KUKA KRL program: makro340.src

&ACCESS RVO2
&COMMENT GREIFER INIT
&PARAM TEMPLATE = C:\KRC\Roboter\Template\makrovorgabe.src
&PARAM TPVW_VERSION = 8.1.8
&PARAM EDITMASK = Makro999[0-999]
DEFFCT INT MAKRO340(ADV :IN)
   ;FOLD Makro Anfang ;%{PSE}%MKUKATPVW
      BOOL ADV
      ; interface to basic routines
      EXT  BAS (BAS_COMMAND  :IN,REAL  :IN )
      ; interface to VW-standard routines
      EXT VW (VW_COMMAND:IN, BOOL: IN, REAL:IN, REAL:IN, REAL:IN, REAL:IN, BOOL :IN, E6POS :IN )
      ; interface select routine
      EXTFCT INT  SELECT (SUBTYPE  :IN,INT  :IN,BOOL  :IN,ARI_TYP  :IN,INT  :IN,BOOL_TYP  :IN,INT  :IN,BOOL  :IN)
      SPS_N=-1
      ;FOLD ;%{H} %MKUKATPVW
      IF VARSTATE ("ADV") <> #INITIALIZED THEN
         ADV=FALSE
      ENDIF
      IF (NOT ADV) THEN
      ;ENDFOLD
   ;ENDFOLD
   ;FOLD -- Greifer Initialisierung -- ;%{E}%MKUKATPVW %CVW_COM %VCOMMENT %P 2:-- Greifer Initialisierung --, 3: VW_COMMENT
   ;ENDFOLD
   ;FOLD -- KS24 -- ;%{E}%MKUKATPVW %CVW_COM %VCOMMENT %P 2:-- KS24 --, 3: VW_COMMENT
   ;ENDFOLD
   ;FOLD -- Version: 01 -- ;%{E}%MKUKATPVW %CVW_COM %VCOMMENT %P 2:-- Version: 01 --, 3: VW_COMMENT
   ;ENDFOLD
   ;FOLD -- Stand: 001 -- ;%{E}%MKUKATPVW %CVW_COM %VCOMMENT %P 2:-- Stand: 001 --, 3: VW_COMMENT
   ;ENDFOLD
   ;FOLD -- letzte Aenderung 11.06.2014 PK -- ;%{E}%MKUKATPVW %CVW_COM %VCOMMENT %P 2:-- letzte Aenderung 11.06.2014 PK --, 3: VW_COMMENT
   ;ENDFOLD
   ;FOLD -- Vorwahl Spanngruppen AUS -- ;%{E}%MKUKATPVW %CVW_COM %VCOMMENT %P 2:-- Vorwahl Spanngruppen AUS --, 3: VW_COMMENT
   ;ENDFOLD
   ;FOLD F1 = AUS ;%{E}%MKUKATPVW %CVW_SPS %VBOASG %P 2:F1 = AUS, 3: BOASG
      $FLAG[1] = FALSE
   ;ENDFOLD
   ;FOLD F2 = AUS ;%{E}%MKUKATPVW %CVW_SPS %VBOASG %P 2:F2 = AUS, 3: BOASG
      $FLAG[2] = FALSE
   ;ENDFOLD
   ;FOLD F3 = AUS ;%{E}%MKUKATPVW %CVW_SPS %VBOASG %P 2:F3 = AUS, 3: BOASG
      $FLAG[3] = FALSE
   ;ENDFOLD
   ;FOLD F4 = AUS ;%{E}%MKUKATPVW %CVW_SPS %VBOASG %P 2:F4 = AUS, 3: BOASG
      $FLAG[4] = FALSE
   ;ENDFOLD
   ;FOLD F5 = AUS ;%{E}%MKUKATPVW %CVW_SPS %VBOASG %P 2:F5 = AUS, 3: BOASG
      $FLAG[5] = FALSE
   ;ENDFOLD
   ;FOLD F6 = AUS ;%{E}%MKUKATPVW %CVW_SPS %VBOASG %P 2:F6 = AUS, 3: BOASG
      $FLAG[6] = FALSE
   ;ENDFOLD
   ;FOLD F7 = AUS ;%{E}%MKUKATPVW %CVW_SPS %VBOASG %P 2:F7 = AUS, 3: BOASG
      $FLAG[7] = FALSE
   ;ENDFOLD
   ;FOLD F8 = AUS ;%{E}%MKUKATPVW %CVW_SPS %VBOASG %P 2:F8 = AUS, 3: BOASG
      $FLAG[8] = FALSE
   ;ENDFOLD
   ;FOLD F9 = AUS ;%{E}%MKUKATPVW %CVW_SPS %VBOASG %P 2:F9 = AUS, 3: BOASG
      $FLAG[9] = FALSE
   ;ENDFOLD
   ;FOLD F10 = AUS ;%{E}%MKUKATPVW %CVW_SPS %VBOASG %P 2:F10 = AUS, 3: BOASG
      $FLAG[10] = FALSE
   ;ENDFOLD
   ;FOLD F11 = AUS ;%{E}%MKUKATPVW %CVW_SPS %VBOASG %P 2:F11 = AUS, 3: BOASG
      $FLAG[11] = FALSE
   ;ENDFOLD
   ;FOLD F12 = AUS ;%{E}%MKUKATPVW %CVW_SPS %VBOASG %P 2:F12 = AUS, 3: BOASG
      $FLAG[12] = FALSE
   ;ENDFOLD
   ;FOLD F13 = AUS ;%{E}%MKUKATPVW %CVW_SPS %VBOASG %P 2:F13 = AUS, 3: BOASG
      $FLAG[13] = FALSE
   ;ENDFOLD
   ;FOLD F14 = AUS ;%{E}%MKUKATPVW %CVW_SPS %VBOASG %P 2:F14 = AUS, 3: BOASG
      $FLAG[14] = FALSE
   ;ENDFOLD
   ;FOLD F15 = AUS ;%{E}%MKUKATPVW %CVW_SPS %VBOASG %P 2:F15 = AUS, 3: BOASG
      $FLAG[15] = FALSE
   ;ENDFOLD
   ;FOLD F16 = AUS ;%{E}%MKUKATPVW %CVW_SPS %VBOASG %P 2:F16 = AUS, 3: BOASG
      $FLAG[16] = FALSE
   ;ENDFOLD
   ;FOLD F17 = AUS ;%{E}%MKUKATPVW %CVW_SPS %VBOASG %P 2:F17 = AUS, 3: BOASG
      $FLAG[17] = FALSE
   ;ENDFOLD
   ;FOLD F18 = AUS ;%{E}%MKUKATPVW %CVW_SPS %VBOASG %P 2:F18 = AUS, 3: BOASG
      $FLAG[18] = FALSE
   ;ENDFOLD
   ;FOLD F19 = AUS ;%{E}%MKUKATPVW %CVW_SPS %VBOASG %P 2:F19 = AUS, 3: BOASG
      $FLAG[19] = FALSE
   ;ENDFOLD
   ;FOLD F20 = AUS ;%{E}%MKUKATPVW %CVW_SPS %VBOASG %P 2:F20 = AUS, 3: BOASG
      $FLAG[20] = FALSE
   ;ENDFOLD
   ;FOLD F21 = AUS ;%{E}%MKUKATPVW %CVW_SPS %VBOASG %P 2:F21 = AUS, 3: BOASG
      $FLAG[21] = FALSE
   ;ENDFOLD
   ;FOLD F22 = AUS ;%{E}%MKUKATPVW %CVW_SPS %VBOASG %P 2:F22 = AUS, 3: BOASG
      $FLAG[22] = FALSE
   ;ENDFOLD
   ;FOLD F23 = AUS ;%{E}%MKUKATPVW %CVW_SPS %VBOASG %P 2:F23 = AUS, 3: BOASG
      $FLAG[23] = FALSE
   ;ENDFOLD
   ;FOLD F58 = AUS ;%{E}%MKUKATPVW %CVW_SPS %VBOASG %P 2:F58 = AUS, 3: BOASG
      $FLAG[58] = FALSE
   ;ENDFOLD
   ;FOLD F60 = AUS ;%{E}%MKUKATPVW %CVW_SPS %VBOASG %P 2:F60 = AUS, 3: BOASG
      $FLAG[60] = FALSE
   ;ENDFOLD
   ;FOLD F61 = AUS ;%{E}%MKUKATPVW %CVW_SPS %VBOASG %P 2:F61 = AUS, 3: BOASG
      $FLAG[61] = FALSE
   ;ENDFOLD
   ; FOLD ;%{H}
   RETURN 1
   ELSE
   RETURN 1
   ENDIF
ENDFCT
; ENDFOLD
